// TIA Portal V17 export
// export: Created 2024-08-09T12:53:20.7660224Z, ExportSetting WithDefaults, DisplayName Totally Integrated Automation Portal, DisplayVersion V17 Update 7, DisplayName TIA Portal Openness, DisplayVersion V17 Update 7, DisplayName TIA Portal Version Control Interface, DisplayVersion V17, DisplayName STEP 7 Professional, DisplayVersion V17 Update 7, DisplayName STEP 7 Safety, DisplayVersion V17 Update 6, DisplayName WinCC Professional, DisplayVersion V17 Update 7
TYPE "S_MODULE_SUIVI_COMMUNTRANS"
// stored: IsFailsafeCompliant false
   STRUCT
      Tab_Lots { ExternalAccessible := 'False'; ExternalVisible := 'False'; ExternalWritable := 'False'} : Array[0.."MAX_LOTS"] of "S_SUIVI_TRANSF";   // Table des zones de suivi lot
      NiPrec { ExternalAccessible := 'False'; ExternalVisible := 'False'; ExternalWritable := 'False'} : USInt;   // No de lot precedent
      IntVideConnue { ExternalAccessible := 'False'; ExternalVisible := 'False'; ExternalWritable := 'False'} : USInt;   // valeur intensite a vide
      Alternance { ExternalAccessible := 'False'; ExternalVisible := 'False'; ExternalWritable := 'False'} : USInt;   // memo alternances diverses (tremie broyeur)
      NbLotsBr { ExternalAccessible := 'False'; ExternalVisible := 'False'; ExternalWritable := 'False'} : USInt;   // Nbr de lots passes sur le broyeur
      NumLot { ExternalAccessible := 'False'; ExternalVisible := 'False'; ExternalWritable := 'False'} : USInt;   // no de lot pour gestion couleurs
   END_STRUCT;
END_TYPE
